PROGRAM FunktionBlockDiagram
VAR
	 Level_INT : INT;
	 Error_INT : INT;
	 Pump_INT : INT;
	 Pump_LIMIT: INT;
END_VAR

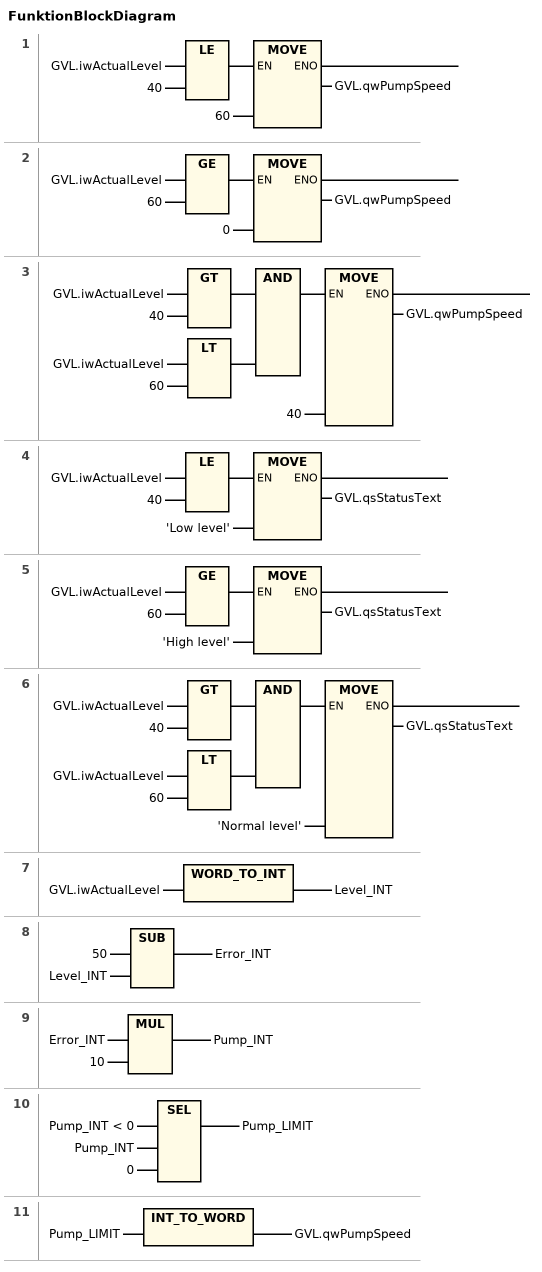
// NETWORK 1
IF GVL.iwActualLevel <= 40 THEN GVL.qwPumpSpeed := 60; END_IF

// NETWORK 2
IF GVL.iwActualLevel >= 60 THEN GVL.qwPumpSpeed := 0; END_IF

// NETWORK 3
IF GVL.iwActualLevel > 40 AND GVL.iwActualLevel < 60 THEN GVL.qwPumpSpeed := 40; END_IF

// NETWORK 4
IF GVL.iwActualLevel <= 40 THEN GVL.qsStatusText := 'Low level'; END_IF

// NETWORK 5
IF GVL.iwActualLevel >= 60 THEN GVL.qsStatusText := 'High level'; END_IF

// NETWORK 6
IF GVL.iwActualLevel > 40 AND GVL.iwActualLevel < 60 THEN GVL.qsStatusText := 'Normal level'; END_IF

// NETWORK 7
Level_INT := WORD_TO_INT(GVL.iwActualLevel);

// NETWORK 8
Error_INT := 50 - Level_INT;

// NETWORK 9
Pump_INT := Error_INT * 10;

// NETWORK 10
Pump_LIMIT := SEL(Pump_INT < 0, Pump_INT, 0);

// NETWORK 11
GVL.qwPumpSpeed := INT_TO_WORD(Pump_LIMIT);

END_PROGRAM

(* stored: Version 1.1.0.1
   POU FunktionBlockDiagram: Id {bb9f87a0-c1f0-406b-9126-1016eb4ae4b7}, SpecialFunc None *)
